TYPE ST_Wago750495_Data :
STRUCT
	//Voltages
	ar_VoltageLN					: ARRAY [0..3] OF REAL;
	ar_VoltageLL					: ARRAY [0..3] OF REAL;
	                            	      
	//Currents 
	ar_CurrentRMS					: ARRAY [0..4] OF REAL;                 	      
	                            	      
	//Power
	ar_ActivePower					: ARRAY [0..3] OF REAL;
	ar_ReactivePower				: ARRAY [0..3] OF REAL;
	ar_ApparentPower				: ARRAY [0..3] OF REAL;                     	      
	
	//Energy
	r_ActiveEnergyTotal				: REAL;
	r_ActiveEnergyImport			: REAL;
	r_ActiveEnergyExport			: REAL;
	r_ReactiveEnergyTotal			: REAL;
	r_ReactiveEnergyInductive		: REAL;
	r_AReactiveEnergyCapacitive		: REAL;
	
	//Frequency
	ar_Frequency					: ARRAY [0..3] OF REAL;
	                        		      
	//Phase Angle 
	ar_PhaseAngle					: ARRAY [0..3] OF REAL;          		      
	                        		      
	//PowerFactor     
	ar_Powerfactor					: ARRAY [0..3] OF REAL;      		      
	
	
END_STRUCT
END_TYPE

(* stored: Version 1.1.0.1, ProductVersion 3.1.4024.12
   DUT ST_Wago750495_Data: Id {cc89ebd2-af3a-4112-b6e9-0c01eea13681} *)
